// TwinCAT 3 PLC project EventLogLib
// Title: Eventlogger Library
// Company: Beckhoff UK
// Author: Chris Knight
// ProjectVersion: 2.1.0.0
// ProgramVersion: 3.1.4026.14
// libraries:
//   Tc2_System, * (Beckhoff Automation GmbH)
//   Tc3_EventLogger, * (Beckhoff Automation GmbH)
// project tree:
//   EventLoggerClass/ I_Message.TcIO, Message.TcPOU, Message_Null.TcPOU

// ---- EventLoggerClass/I_Message.TcIO
INTERFACE I_Message

METHOD Send : HRESULT
VAR_INPUT
	Message : T_MaxString;
END_VAR
END_METHOD

END_INTERFACE

// ---- EventLoggerClass/Message.TcPOU
FUNCTION_BLOCK Message IMPLEMENTS I_Message
VAR_INPUT
END_VAR
VAR_OUTPUT
END_VAR
VAR
    fbMsg : FB_TcMessage; 
	_loggerLevel : TcEventSeverity := TcEventSeverity.Info;
END_VAR

{analysis -2}

//FB_Init is always available implicitly and it is used primarily for initialization.
//The return value is not evaluated. For a specific influence, you can also declare the
//methods explicitly and provide additional code there with the standard initialization
//code. You can evaluate the return value.
METHOD FB_Init: BOOL
VAR_INPUT
    bInitRetains: BOOL; // TRUE: the retain variables are initialized (reset warm / reset cold)
    bInCopyCode: BOOL;  // TRUE: the instance will be copied to the copy code afterward (online change)   
END_VAR
THIS^.fbMsg.CreateEx(TC_Events.Tracing.LogMessage, 0);
END_METHOD

METHOD PUBLIC Send : HRESULT
VAR_INPUT
	Message : T_MaxString;
END_VAR
VAR
	CreateString : HRESULT;
	AddStringResult : I_TcArguments;
	SendResult : HRESULT;
	ReleaseResult : HRESULT;
END_VAR
fbMsg.ipArguments.Clear();
fbMsg.ipArguments.AddString(Message);
SendResult := THIS^.fbMsg.Send(0);
IF SendResult = S_OK THEN
	Send := 1;
ELSE
	Send := -1;
END_IF
END_METHOD

END_FUNCTION_BLOCK

// ---- EventLoggerClass/Message_Null.TcPOU
FUNCTION_BLOCK Message_Null IMPLEMENTS I_Message
VAR
END_VAR

METHOD Send : HRESULT
VAR_INPUT
	Message	: T_MaxString;
END_VAR
END_METHOD

END_FUNCTION_BLOCK
